(* IEC 61131-3 sources: JaccoSigma/tempclass/Class/FDD3000_ParametersFileRam, 1 file *)

(* ---- FDD3000_ParametersFileRam.st ---- *)
#define FDD3000_PARAMETERSFILERAM_AMOUNT_SERVERS   21 //amount of servers of this class

(*!
<Class
	Name               = "FDD3000_ParametersFileRam"
	Revision           = "1.0"
	RealtimeTask       = "false"
	CyclicTask         = "false"
	BackgroundTask     = "false"
	Sigmatek           = "true"
	OSInterface        = "false"
	HighPriority       = "false"
	Automatic          = "false"
	UpdateMode         = "Prescan"
	SharedCommandTable = "true"
	Objectsize         = "(810,600)">
	<Channels>
		<Server Name="AccRate" Visualized="true" Initialize="false" WriteProtected="false" Retentive="File" Comment="Parameter 02.011  Acceleration Rate 1 &#13;&#10;Short description: Defines the acceleration rate present in acceleration rate 1 as [0.0 s].&#13;&#10;"/>
		<Server Name="ClassSvr" Visualized="false" Initialize="false" WriteProtected="true" Retentive="false" Comment="Has no function."/>
		<Server Name="CurrentAtMaximumDeadTime" Visualized="true" Initialize="false" WriteProtected="false" Retentive="File" Comment="OpenLoop Current At Maximum Deadtime Compensation (05.060)&#13;&#10;Short description Current at which maximum deadtime compensation is applied as [0.00 %]&#13;&#10;Read Only"/>
		<Server Name="CurrentLoopKiGain" Visualized="true" Initialize="false" WriteProtected="false" Retentive="File" Comment="RFC-A Current Loop Ki Gain 04.014&#13;&#10;Short description: Defines the current loop controller integral gain as [0.000]"/>
		<Server Name="CurrentLoopKPGain" Visualized="true" Initialize="false" WriteProtected="false" Retentive="File" Comment="RFC-A Current Loop Kp Gain 04.013&#13;&#10;Short description: Defines the current loop controller proportional gain as [0.00]."/>
		<Server Name="DecRate" Visualized="true" Initialize="false" WriteProtected="false" Retentive="File" Comment="Parameter 02.021  Deceleration Rate 1 &#13;&#10;Short description: Defines the deceleration rate present in deceleration rate 1 as [0.0 s].&#13;&#10;"/>
		<Server Name="LowFrequencyVoltageBoost" Visualized="true" Initialize="false" WriteProtected="false" Retentive="File" Comment="Parameter 05.015  Low Frequency Voltage Boost &#13;&#10;Short description: Defines the level of voltage boost &#13;&#10;at 0Hz when using a fixed V to F relationship as [0.0 %].  &#13;&#10;"/>
		<Server Name="MaximumDeadTimeComp" Visualized="true" Initialize="false" WriteProtected="false" Retentive="File" Comment="OpenLoop Maximum Deadtime compensation 05.059&#13;&#10;Short description: Maximum Deadtime Compensation  as [0.000 µs]&#13;&#10;Read Only"/>
		<Server Name="MaxRefClamp" Visualized="true" Initialize="false" WriteProtected="false" Retentive="File" Comment="Parameter 01.006  Maximum Reference Clamp &#13;&#10;Short description: Defines the maximum value for the reference as [0.00 Hz].&#13;&#10;"/>
		<Server Name="MinRefClamp" Visualized="true" Initialize="false" WriteProtected="false" Retentive="File" Comment="Parameter 01.007  Minimum Reference Clamp &#13;&#10;Short description: Defines the minimum value for the reference  as [0.00 Hz].&#13;&#10;"/>
		<Server Name="MotorRatedCurrent" Visualized="true" Initialize="false" WriteProtected="false" Retentive="File" Comment="Parameter 05.007  Motor Rated Current &#13;&#10;Short description: Set to the rated current rated of the motor as [0.00 A].&#13;&#10;"/>
		<Server Name="MotorRatedFrequency" Visualized="true" Initialize="false" WriteProtected="false" Retentive="File" Comment="Parameter 05.006  Motor Rated Frequency &#13;&#10;Short description: Set to the rated frequency of the motor as [0.00 Hz]. &#13;&#10;"/>
		<Server Name="MotorRatedPowerFactor" Visualized="true" Initialize="false" WriteProtected="false" Retentive="File" Comment="Parameter 05.010  Motor Rated Power Factor &#13;&#10;Short description: Set to the rated power factor of the motor as [0.00].  &#13;&#10;This value can be measured by the drive during a rotating autotune.&#13;&#10;"/>
		<Server Name="MotorRatedSpeed" Visualized="true" Initialize="false" WriteProtected="false" Retentive="File" Comment="Parameter 05.008  Motor Rated Speed &#13;&#10;Short description: Set to the rated speed of the motor as [0.0 rpm]. &#13;&#10;"/>
		<Server Name="MotorRatedVoltage" Visualized="true" Initialize="false" WriteProtected="false" Retentive="File" Comment="Parameter 05.009  Motor Rated Voltage &#13;&#10;Short description: Set to the rated voltage of the motor as [V]. &#13;&#10;"/>
		<Server Name="SaturationBreakpoint1" Visualized="true" Initialize="false" WriteProtected="false" Retentive="File" Comment="RFC-A motor saturation breakpoints Pr 05.029 &#13;&#10;Short description: Defines Saturation Breakpoint 1 within &#13;&#10;the saturation characteristic as [0.0 %]. &#13;&#10;"/>
		<Server Name="SaturationBreakpoint2" Visualized="true" Initialize="false" WriteProtected="false" Retentive="File" Comment="RFC-A motor saturation breakpoints Pr 05.062&#13;&#10;Short description: Defines Saturation Breakpoint 2 within &#13;&#10;the saturation characteristic as [0.0 %]. "/>
		<Server Name="SaturationBreakpoint3" Visualized="true" Initialize="false" WriteProtected="false" Retentive="File" Comment="RFC-A motor saturation breakpoints Pr 05.030&#13;&#10;Short description: Defines Saturation Breakpoint 3 within &#13;&#10;the saturation characteristic as [0.0 %]. "/>
		<Server Name="SaturationBreakpoint4" Visualized="true" Initialize="false" WriteProtected="false" Retentive="File" Comment="RFC-A motor saturation breakpoints Pr 05.063&#13;&#10;Short description: Defines Saturation Breakpoint 4 within &#13;&#10;the saturation characteristic as [0.0 %]. "/>
		<Server Name="StatorInductance" Visualized="true" Initialize="false" WriteProtected="false" Retentive="File" Comment="OpenLoop / RFC-A Stator Inductance 05.025&#13;&#10;Short description: Defines the inductance of the motor stator as [0.00 mH]."/>
		<Server Name="StatorResistance" Visualized="true" Initialize="false" WriteProtected="false" Retentive="File" Comment="OpenLoop / RFC-A Stator Resistance 05.017&#13;&#10;Short description: Defines the resistance of the motor stator as [0.0000 ohm]"/>
		<Server Name="TransientInductance" Visualized="true" Initialize="false" WriteProtected="false" Retentive="File" Comment="OpenLoop / RFC-A Transient Inductance 05.024&#13;&#10;Short description: Defines the inducatance of the transient &#13;&#10;components in the motor stator as [0.000 mH] "/>
	</Channels>
	<Separators>
		<Servers>
			<SepChn Position="19"/>
			<SepChn Position="16"/>
			<SepChn Position="12"/>
			<SepChn Position="1"/>
		</Servers>
	</Separators>
	<RevDoku>
		<Owner Company="Sigmatek" Author="PieSte"/>
		<Dokumentation Revision="1.0" Date="02.02.2021" Author="ZoePat" Company="Sigmatek" Description="first library version"/>
	</RevDoku>
</Class>
*)
FDD3000_ParametersFileRam : CLASS
  //Servers:
	ClassSvr 	: SvrChCmd_DINT;
	MaxRefClamp 	: SvrCh_DINT;
	MinRefClamp 	: SvrCh_DINT;
	AccRate 	: SvrCh_DINT;
	DecRate 	: SvrCh_DINT;
	MotorRatedCurrent 	: SvrCh_DINT;
	MotorRatedSpeed 	: SvrCh_DINT;
	MotorRatedVoltage 	: SvrCh_DINT;
	MotorRatedPowerFactor 	: SvrCh_DINT;
	MotorRatedFrequency 	: SvrCh_DINT;
	LowFrequencyVoltageBoost 	: SvrCh_DINT;
	StatorResistance 	: SvrCh_DINT;
	TransientInductance 	: SvrCh_DINT;
	StatorInductance 	: SvrCh_DINT;
	MaximumDeadTimeComp 	: SvrCh_DINT;
	CurrentAtMaximumDeadTime 	: SvrCh_DINT;
	CurrentLoopKPGain 	: SvrCh_DINT;
	CurrentLoopKiGain 	: SvrCh_DINT;
	SaturationBreakpoint1 	: SvrCh_DINT;
	SaturationBreakpoint3 	: SvrCh_DINT;
	SaturationBreakpoint2 	: SvrCh_DINT;
	SaturationBreakpoint4 	: SvrCh_DINT;
  //Clients:
  //Variables:
  //Functions:
  //Tables:
	FUNCTION @STD
		VAR_OUTPUT
			ret_code	: CONFSTATES;
		END_VAR;
	FUNCTION GLOBAL TAB @CT_;
END_CLASS;
